PROGRAM PRG_1_PlcTask
VAR
END_VAR

PRG_MR1L1_HOMS();

END_PROGRAM

(* stored: Version 1.1.0.1, ProductVersion 3.1.4022.18
   POU PRG_1_PlcTask: Id {e42871bb-98ad-406e-a48f-123eec67eb14}, SpecialFunc None *)
